(* IEC 61131-3 sources: Generators/test, 4 files *)

(* ---- dummy.st ---- *)
NAMESPACE Simatic.Ax.Generators
{TestFixture}
CLASS MyTestFixture
    {Test}
    METHOD PUBLIC MyTestMethod
        AxUnit.Assert.Equal(TRUE, TRUE);
    END_METHOD
END_CLASS
END_NAMESPACE

(* ---- OnDelayMockWithTwoTimers.st ---- *)
NAMESPACE Simatic.Ax.Mocks
    /// This Mock can be used in Classes/FunctionBlocks where are two OnDelay instances are used
    {axcode:docs-v0:@simatic-ax/generators:OnDelayMockWithTwoTimers.md}
    FUNCTION_BLOCK OnDelayMock2Timer
        VAR_INPUT
            /// Signal to be monitored.
            signal: BOOL;
            /// Duration of the delay.
            duration: LTIME;
        END_VAR

        VAR_OUTPUT
            /// Operand that is set after the delay.
            output: BOOL;
            /// Current elapsed time.
            elapsedTime: LTIME;
        END_VAR

        VAR_TEMP
            state : REF_TO OnDelayMockState;
        END_VAR

        state ?= AxUnit.Mocking.GetPayload();
        output := TRUE;

        IF (signal = FALSE) THEN
            output := FALSE;
        ELSE
            IF duration = T#1s THEN
                output := state^.StatusTimer1;
            END_IF;
            IF duration = T#2s THEN
                output := state^.StatusTimer2 ;
            END_IF;
        END_IF;

    END_FUNCTION_BLOCK

    /// The returned states for the Timer1 and Timer2
    {axcode:docs-v0:@simatic-ax/generators:OnDelayMockWithTwoTimers.md}
    CLASS OnDelayMockState IMPLEMENTS AxUnit.Mocking.IPayload
        VAR PUBLIC
            StatusTimer1 : BOOL;
            StatusTimer2 : BOOL;
        END_VAR
    END_CLASS
END_NAMESPACE

(* ---- test.st ---- *)
USING AxUnit.Assert;
USING Simatic.Ax.Generators;

NAMESPACE Simatic.Ax.Library
    {TestFixture}
    CLASS MyTestFixture
        VAR
            o : PulseGenerator;
        END_VAR

        {Test}
        METHOD PUBLIC MyTestMethod
            o.Execute();
            ; // AxUnit.Assert.Equal(expected := y, actual := x);
        END_METHOD
    END_CLASS
END_NAMESPACE

(* ---- TestOnCycle.st ---- *)
USING Simatic.Ax.Generators;
USING Simatic.Ax.Mocks;

NAMESPACE Simatic.Ax.Generators.Test
    {TestFixture}
    CLASS TestActiveWait
        VAR
                _state : OnDelayMockState;
                testInstance : PulseGenerator;
        END_VAR

        {Test}
        METHOD PUBLIC Test_One_Clock_Cycle_Expect_True_False_True
            VAR_TEMP
                res : BOOL;
            END_VAR
            testInstance.PulseTime := T#1s; // give the mocked timer an value to distiguish in the mock
            testInstance.PauseTime := T#2s;

            // Initial state --> Clock returns true, no timer is running
            _state.StatusTimer1 := FALSE;
            _state.StatusTimer2 := FALSE;

            AxUnit.Mocking.Mock('System.Timer.OnDelay', NAME_OF(OnDelayMock2Timer), THIS._state);
            testInstance.Execute();
            res := testInstance.Q();
            AxUnit.Assert.Equal(TRUE, res);

            // second cycle --> Clock returns still true
            testInstance.Execute();

            res := testInstance.Q();
            AxUnit.Assert.Equal(TRUE, res);

            // third cycle --> PulseTime has elapsed --> Clock returns false
            _state.StatusTimer1 := TRUE;
            _state.StatusTimer2 := FALSE;
            testInstance.Execute();
            res := testInstance.Q();
            AxUnit.Assert.Equal(FALSE, res);

            // 4th Cycle  --> Clock returns still false. PauseTimer is running but is not elapsed
            _state.StatusTimer1 := FALSE;
            _state.StatusTimer2 := FALSE;
            testInstance.Execute();
            res := testInstance.Q();
            AxUnit.Assert.Equal(FALSE, res);

            // 5th cycle --> PauseTime has elapsed --> Clock returns false
            _state.StatusTimer1 := FALSE;
            _state.StatusTimer2 := TRUE;
            testInstance.Execute();
            res := testInstance.Q();
            AxUnit.Assert.Equal(TRUE, res);
        END_METHOD

    END_CLASS

END_NAMESPACE
